(* CODESYS project Raspberry.project

Project tree, tasks and I/O mapping:
  Device : CODESYS Control for Raspberry Pi, 3S - Smart Software Solutions GmbH, version 3.5.7.0
    application Application
      libraries: Standard, * (System)
      task MainTask (cyclic, interval t#20ms, priority 1) calls PLC_PRG, LED_UpDown
      task VISU_TASK (cyclic, interval 100 ms, priority 30) calls VisuElems.Visu_Prg
      program PLC_PRG [ST]: UpdateLed, UpdateLedStrip
      visualisation MainPage
      data type LED_Strip
      data type LED
      visualisation Led
      program LED_UpDown [FBD]
      global variables GVL
    SoftMotion General Axis Pool
    GPIOs : GPIOs B+/Pi2, 3S - Smart Software Solutions GmbH, version 1.1.1.0
        unmapped channels: digital inputs (GPIO0..GPIO31), digital outputs (GPIO0..GPIO31)
    Camera device
      <Empty>
    ModbusConfig : Ethernet, 3S - Smart Software Solutions GmbH, version 3.5.7.0
        settings: NetworkInterfaceName = 'ether0'
      Modbus_TCP_Master : Modbus TCP Master, 3S - Smart Software Solutions GmbH, version 3.5.6.0
          settings: AutoReconnect = TRUE
        Makeblock : Modbus TCP Slave, 3S - Smart Software Solutions GmbH, version 3.5.7.0
            settings: IPAddress = [192, 168, 0, 40]; Channel 0.Function Code = 15; Channel 0.Read Offset = 0; Channel 0.Read Length = 0; Channel 0.Write Offset = 16#0000; Channel 0.Write Length = 8; Channel 0.Cycle Time = 50; Channel 3.Function Code = 16; Channel 3.Read Offset = 0; Channel 3.Read Length = 0; Channel 3.Write Offset = 16#0000; Channel 3.Write Length = 15; Channel 3.Cycle Time = 100; Channel 2.Function Code = 1; Channel 2.Read Offset = 16#0000; Channel 2.Read Length = 8; Channel 2.Write Offset = 0; Channel 2.Write Length = 0; Channel 2.Cycle Time = 50
            unmapped channels: Channel 0, Channel 3, Channel 2
    I²C
    SPI
    Onewire
  text list GlobalTextList
  GlobalImagePool
*)

// Device/Application/LED_Strip
TYPE LED_Strip :
STRUCT
	LEDs:ARRAY [1..15] OF LED; 
END_STRUCT
END_TYPE

// Device/Application/LED
TYPE LED :
	STRUCT
		TurnOn:BOOL;
		Green:BOOL;
		Red:BOOL;
		Yellow:BOOL;
		Blue:BOOL;
		Grey:BOOL;
		ColorReg:INT;
	END_STRUCT
END_TYPE

// Device/Application/GVL
VAR_GLOBAL
	LedStrip1: LED_Strip;
END_VAR

// Device/Application/PLC_PRG
PROGRAM PLC_PRG
VAR
	Sensor1: BOOL; 				// Line follower sensor 1
	Sensor2: BOOL; 				// Line follower sensor 2
	LedStripRed: BOOL; 			// Turn the LED strip Red
	LedStripGreen: BOOL; 		// Turn the LED strip Green
	
	PushButton1: BOOL := FALSE;;			// Push button in GUI
	PushButton2: BOOL := FALSE;;			// Push button in GUI
	PushButtonNightRider: BOOL := FALSE;	// Push button in GUI

	Pulse:BOOL := FALSE;
END_VAR

// Input Mapping
Sensor1:=%IX0.0;
Sensor2:=%IX0.1;

// Logic
LedStripRed := Sensor1 OR PushButton1;
LedStripGreen := Sensor2 OR PushButton2;

IF NOT PushButtonNightRider THEN
	IF LedStripGreen THEN
		UpdateLedStrip(TRUE, TRUE, FALSE, FALSE, FALSE, LedStrip := LedStrip1);
	ELSIF LedStripRed THEN
		UpdateLedStrip(TRUE, FALSE, TRUE, FALSE, FALSE, LedStrip := LedStrip1);
	ELSE
		UpdateLedStrip(FALSE, TRUE, FALSE, FALSE, FALSE, LedStrip := LedStrip1);
	END_IF
END_IF

%QW1:=INT_TO_WORD(LedStrip1.LEDs[1].ColorReg);
%QW2:=INT_TO_WORD(LedStrip1.LEDs[2].ColorReg);
%QW3:=INT_TO_WORD(LedStrip1.LEDs[3].ColorReg);
%QW4:=INT_TO_WORD(LedStrip1.LEDs[4].ColorReg);
%QW5:=INT_TO_WORD(LedStrip1.LEDs[5].ColorReg);
%QW6:=INT_TO_WORD(LedStrip1.LEDs[6].ColorReg);
%QW7:=INT_TO_WORD(LedStrip1.LEDs[7].ColorReg);
%QW8:=INT_TO_WORD(LedStrip1.LEDs[8].ColorReg);
%QW9:=INT_TO_WORD(LedStrip1.LEDs[9].ColorReg);
%QW10:=INT_TO_WORD(LedStrip1.LEDs[10].ColorReg);
%QW11:=INT_TO_WORD(LedStrip1.LEDs[11].ColorReg);
%QW12:=INT_TO_WORD(LedStrip1.LEDs[12].ColorReg);
%QW13:=INT_TO_WORD(LedStrip1.LEDs[13].ColorReg);
%QW14:=INT_TO_WORD(LedStrip1.LEDs[14].ColorReg);
%QW15:=INT_TO_WORD(LedStrip1.LEDs[15].ColorReg);

METHOD UpdateLed
VAR_INPUT
	EN:BOOL;
	index:INT := 1;
	State:BOOL;
	Green:BOOL;
	Red:BOOL;
	Yellow:BOOL;
	Blue:BOOL;
END_VAR

VAR_IN_OUT
	Led: LED_Strip;
END_VAR
IF EN THEN
	
	IF index < 1 THEN 
		index:=1;
	ELSIF index > 15 THEN
		index:=15;
	END_IF
	
	Led.LEDs[index].TurnOn := State;
	
	IF Green THEN
		Led.LEDs[index].Green := FALSE;
		Led.LEDs[index].Red := TRUE;
		Led.LEDs[index].Yellow := TRUE;
		Led.LEDs[index].Blue := TRUE;
		Led.LEDs[index].ColorReg := 1;
	ELSIF Red THEN
		Led.LEDs[index].Green := TRUE;
		Led.LEDs[index].Red := FALSE;
		Led.LEDs[index].Yellow := TRUE;
		Led.LEDs[index].Blue := TRUE;
		Led.LEDs[index].ColorReg := 2;
	ELSIF Yellow THEN
		Led.LEDs[index].Green := TRUE;
		Led.LEDs[index].Red := TRUE;
		Led.LEDs[index].Yellow := FALSE;
		Led.LEDs[index].Blue := TRUE;
		Led.LEDs[index].ColorReg := 3;
	ELSIF Blue THEN
		Led.LEDs[index].Green := TRUE;
		Led.LEDs[index].Red := TRUE;
		Led.LEDs[index].Yellow := TRUE;
		Led.LEDs[index].Blue := FALSE;
		Led.LEDs[index].ColorReg := 4;
	END_IF
	
	IF NOT State THEN
		Led.LEDs[index].ColorReg := 0;
	END_IF
END_IF
END_METHOD

METHOD UpdateLedStrip
VAR_INPUT
	State:BOOL;
	Green:BOOL;
	Red:BOOL;
	Yellow:BOOL;
	Blue:BOOL;
END_VAR

VAR
	iCounter: INT;
END_VAR
VAR_IN_OUT
	LedStrip: LED_Strip;
END_VAR

FOR iCounter := 1 TO 15 BY 1 DO
	updateLed(TRUE,iCounter,State,Green,Red,Yellow,Blue, Led := LedStrip);
END_FOR;
END_METHOD

END_PROGRAM

// Device/Application/LED_UpDown
PROGRAM LED_UpDown
VAR
	Green:BOOL;
	Red:BOOL;
	Yellow:BOOL;
	Blue:BOOL:=TRUE;
	currentLED: INT:=1;
	UpperLimit: BOOL := FALSE;
	NegPulse: BOOL;
	Pulse100ms: BOOL;
	LowerLimit: BOOL;
	Up: BOOL := TRUE;
	
	CTUD_0: CTUD;
	TP_0: TP;
	R_TRIG_0: R_TRIG;
	R_TRIG_1: R_TRIG;
	RTC_0: RTC;
	TP_1: TP;
	SR_0: SR;
END_VAR
VAR // added by the converter: edge detectors and wires of the graphical bodies
    _ft1 : F_TRIG;
END_VAR

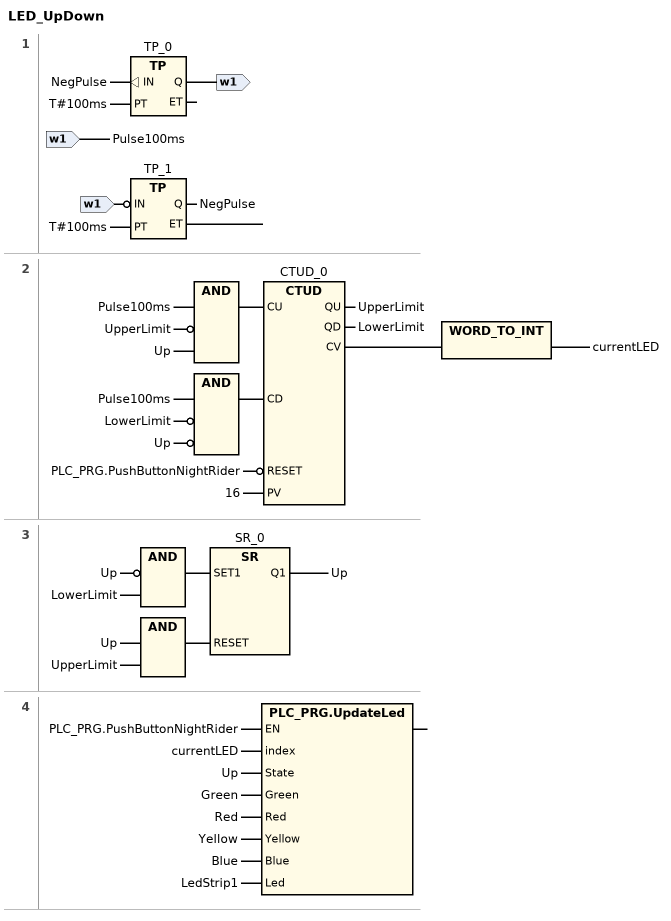
// NETWORK 1
_ft1(CLK := NegPulse);
TP_0(IN := _ft1.Q, PT := T#100ms); // TP
Pulse100ms := TP_0.Q;
TP_1(IN := NOT TP_0.Q, PT := T#100ms, Q => NegPulse); // TP

// NETWORK 2
CTUD_0(
    CU := Pulse100ms AND NOT UpperLimit AND Up,
    CD := Pulse100ms AND NOT LowerLimit AND NOT Up,
    RESET := NOT PLC_PRG.PushButtonNightRider,
    PV := 16,
    QU => UpperLimit,
    QD => LowerLimit); // CTUD
currentLED := WORD_TO_INT(CTUD_0.CV);

// NETWORK 3
SR_0(SET1 := NOT Up AND LowerLimit, RESET := Up AND UpperLimit); // SR
Up := SR_0.Q1;

// NETWORK 4
PLC_PRG.UpdateLed(EN := PLC_PRG.PushButtonNightRider, index := currentLED, State := Up, Green := Green, Red := Red, Yellow := Yellow, Blue := Blue, Led := LedStrip1);

END_PROGRAM

// Device/Application/MainPage
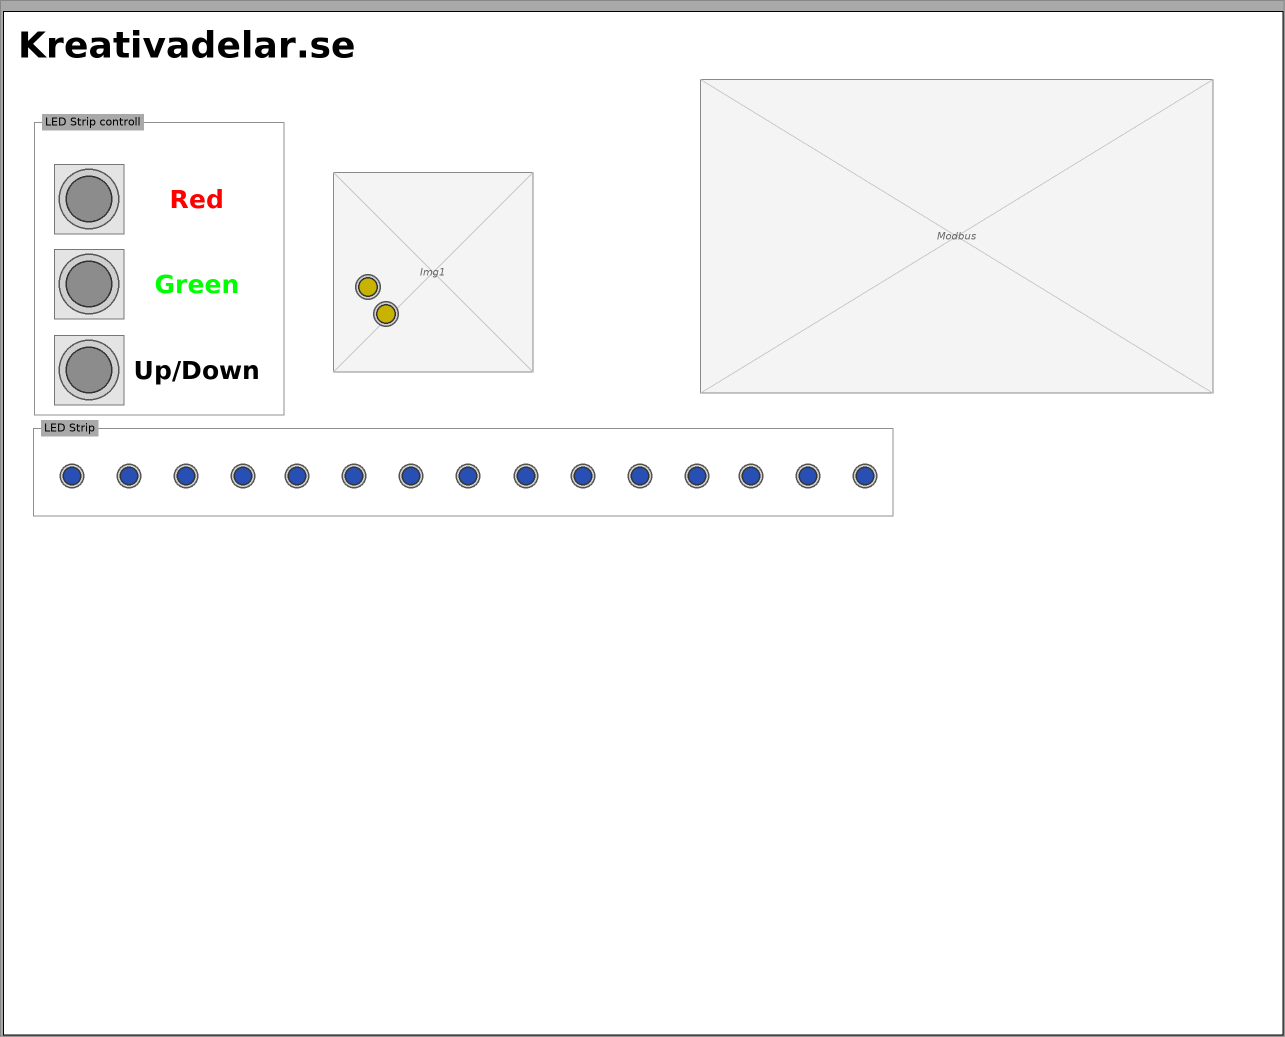
VISUALIZATION MainPage  // 1285x1037
    Rectangle (3,11 1280x1024)
    GroupBox (33,420 860x96), "LED Strip"
        Frame (25,42 30x30)
            shows Led(Led := LedStrip1.LEDs[1])
        Frame (82,42 30x30)
            shows Led(Led := LedStrip1.LEDs[2])
        Frame (139,42 30x30)
            shows Led(Led := LedStrip1.LEDs[3])
        Frame (196,42 30x30)
            shows Led(Led := LedStrip1.LEDs[4])
        Frame (250,42 30x30)
            shows Led(Led := LedStrip1.LEDs[5])
        Frame (307,42 30x30)
            shows Led(Led := LedStrip1.LEDs[6])
        Frame (364,42 30x30)
            shows Led(Led := LedStrip1.LEDs[7])
        Frame (421,42 30x30)
            shows Led(Led := LedStrip1.LEDs[8])
        Frame (479,42 30x30)
            shows Led(Led := LedStrip1.LEDs[9])
        Frame (536,42 30x30)
            shows Led(Led := LedStrip1.LEDs[10])
        Frame (593,42 30x30)
            shows Led(Led := LedStrip1.LEDs[11])
        Frame (650,42 30x30)
            shows Led(Led := LedStrip1.LEDs[12])
        Frame (704,42 30x30)
            shows Led(Led := LedStrip1.LEDs[13])
        Frame (761,42 30x30)
            shows Led(Led := LedStrip1.LEDs[14])
        Frame (818,42 30x30)
            shows Led(Led := LedStrip1.LEDs[15])
    Group (333,172 200x200)
        Image (0,0 200x200), image: Img1
        Lamp1 (20,100 30x30), variable: PLC_PRG.Sensor1, style: Lamp-Lamp1-Yellow
        Lamp1 (38,127 30x30), variable: PLC_PRG.Sensor2, style: Lamp-Lamp1-Yellow
    GroupBox (34,114 250x301), "LED Strip controll"
        PushSwitch (20,221 70x70), variable: PLC_PRG.PushButtonNightRider, behaviour: TOGGLE, style: Switch-PushSwitch-Gray
        Label (88,60 150x50), "Red"
        Label (88,145 150x50), "Green"
        PushSwitch (20,135 70x70), variable: PLC_PRG.PushButton2, behaviour: TOGGLE, style: Switch-PushSwitch-Gray
        PushSwitch (20,50 70x70), variable: PLC_PRG.PushButton1, behaviour: TOGGLE, style: Switch-PushSwitch-Gray
        Label (88,231 150x50), "Up/Down"
    Label (15,30 400x30), "Kreativadelar.se"
    Image (700,79 513x314), image: Modbus
END_VISUALIZATION

// Device/Application/Led
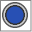
VISUALIZATION Led  // 32x32
VAR_IN_OUT
	Led:LED;
END_VAR
    Lamp1 (0,0 30x30), variable: Led.TurnOn, invisible if: Led.Green, style: Lamp-Lamp1-Green
    Lamp1 (0,0 30x30), variable: Led.TurnOn, invisible if: Led.Red, style: Lamp-Lamp1-Red
    Lamp1 (0,0 30x30), variable: Led.TurnOn, invisible if: Led.Yellow, style: Lamp-Lamp1-Yellow
    Lamp1 (0,0 30x30), variable: Led.TurnOn, invisible if: Led.Blue, style: Lamp-Lamp1-Blue
END_VISUALIZATION
